// TIA Portal V16 export
// export: Created 2023-03-29T11:03:17.6756957Z, ExportSetting WithDefaults, DisplayName Totally Integrated Automation Portal, DisplayVersion V16 Update 6, DisplayName TIA Portal Version Control Interface, DisplayVersion V16 Update 2, DisplayName TIA Portal Openness, DisplayVersion V16 Update 6, DisplayName STEP 7 Professional, DisplayVersion V16 Update 6, DisplayName STEP 7 Safety, DisplayVersion V16, DisplayName WinCC Advanced, DisplayVersion V16 Update 6
ORGANIZATION_BLOCK "Startup"   // OB100, LAD, Startup
TITLE = "Complete Restart"
{ S7_Optimized_Access := 'TRUE' }
VERSION : 0.1
// Zasuwa status aut. zamknięta= 35980
// Zasuwa status aut. otwarta=34438
// stored: AutoNumber true, IsIECCheckEnabled false, SetENOAutomatically false
   VAR_INPUT
      LostRetentive : Bool;   // True if retentive data are lost
      LostRTC : Bool;   // True if date and time are lost
   END_VAR
BEGIN

REGION Network 1: znacznik powrotu zasilania
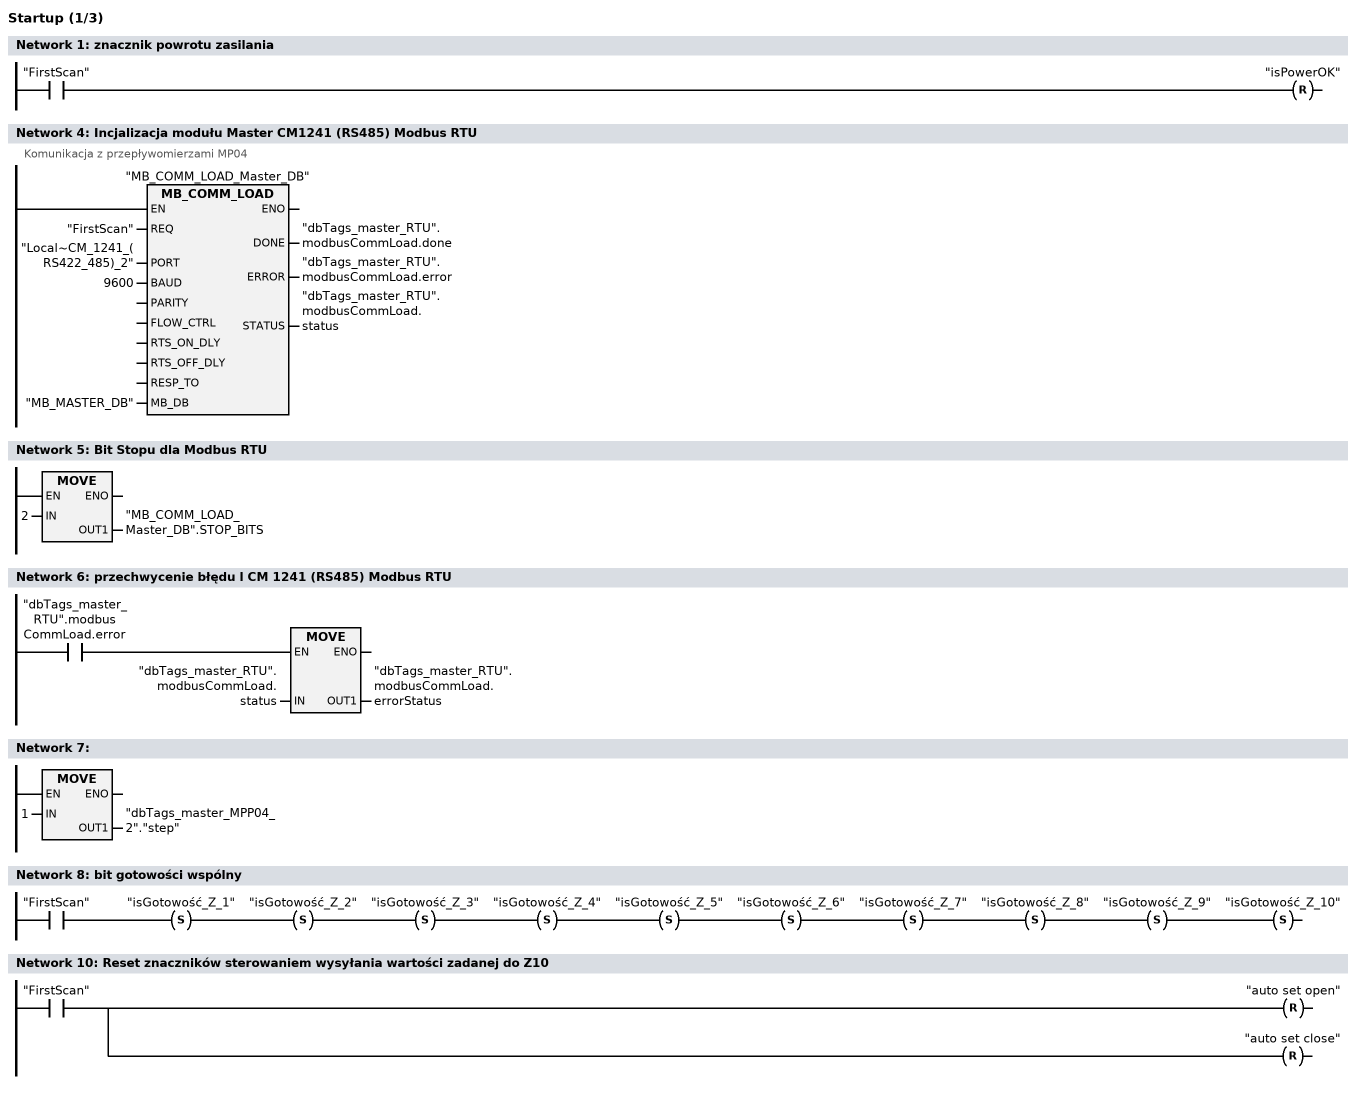
   RUNG wire#powerrail
      Contact( "FirstScan" )
      R_Coil( "isPowerOK" )
   END_RUNG
   // the same network as SCL:
   IF "FirstScan" THEN "isPowerOK" := FALSE; END_IF;
END_REGION

REGION Network 2 (SCL): konfiguracja filtru Kalmana
   IF "FirstScan" THEN //w pierwszym cyklu sterownika
     FOR "I" := 0 TO 3 DO
       "KALMAN_DB".kalman_K["I"] := 0.0;
       "KALMAN_DB".kalman_R["I"] := 0.001;  //niepewność pomiaru
       "KALMAN_DB".kalman_Q["I"] := 0.00001;  //niepewność procesu
       "KALMAN_DB".kalman_P["I"] := 1.0;
     END_FOR;        //parametry R i Q można dobrać osobno dla każdego kanału
   END_IF;           //zostaje wykonana inicjalizacja wszystkich 5 torów analogowych
END_REGION

REGION Network 3 (SCL): Kasowanie alarmów
   "dbtags_Sterowanie".HMI.resetScreen_1 := TRUE;
   "dbtags_Sterowanie".HMI.resetScreen_5 := TRUE;
   "dbtags_Sterowanie".HMI.resetScreen_4 := TRUE;
   "dbtags_Sterowanie".HMI.resetScreen_3 := TRUE;
   "dbtags_Sterowanie".HMI.resetScreen_2 := TRUE;
END_REGION

REGION Network 4: Incjalizacja modułu Master CM1241 (RS485) Modbus RTU
   // Komunikacja z przepływomierzami MP04
   RUNG wire#powerrail
      "MB_COMM_LOAD_Master_DB".MB_COMM_LOAD(REQ := "FirstScan", PORT := "Local~CM_1241_(RS422_485)_2", BAUD := 9600, PARITY :=, FLOW_CTRL :=, RTS_ON_DLY :=, RTS_OFF_DLY :=, RESP_TO :=, MB_DB := "MB_MASTER_DB", DONE => "dbTags_master_RTU".modbusCommLoad.done, ERROR => "dbTags_master_RTU".modbusCommLoad.error, STATUS => "dbTags_master_RTU".modbusCommLoad.status)
   END_RUNG
   // the same network as SCL:
   "MB_COMM_LOAD_Master_DB"(REQ := "FirstScan",   // MB_COMM_LOAD
                           PORT := "Local~CM_1241_(RS422_485)_2",
                           BAUD := 9600,
                           MB_DB := "MB_MASTER_DB",
                           DONE => "dbTags_master_RTU".modbusCommLoad.done,
                           ERROR => "dbTags_master_RTU".modbusCommLoad.error,
                           STATUS => "dbTags_master_RTU".modbusCommLoad.status);
END_REGION

REGION Network 5: Bit Stopu dla Modbus RTU
   RUNG wire#powerrail
      Move(in := 2, out1 => "MB_COMM_LOAD_Master_DB".STOP_BITS)
   END_RUNG
   // the same network as SCL:
   "MB_COMM_LOAD_Master_DB".STOP_BITS := 2;
END_REGION

REGION Network 6: przechwycenie błędu l CM 1241 (RS485) Modbus RTU
   RUNG wire#powerrail
      Contact( "dbTags_master_RTU".modbusCommLoad.error )
      { S7_GenerateENO := "TRUE" } Move(in := "dbTags_master_RTU".modbusCommLoad.status, out1 => "dbTags_master_RTU".modbusCommLoad.errorStatus)
   END_RUNG
   // the same network as SCL:
   IF "dbTags_master_RTU".modbusCommLoad.error THEN
       "dbTags_master_RTU".modbusCommLoad.errorStatus := "dbTags_master_RTU".modbusCommLoad.status;
   END_IF;
END_REGION

REGION Network 7
   RUNG wire#powerrail
      Move(in := 1, out1 => "dbTags_master_MPP04_2"."step")
   END_RUNG
   // the same network as SCL:
   "dbTags_master_MPP04_2"."step" := 1;
END_REGION

REGION Network 8: bit gotowości wspólny
   RUNG wire#powerrail
      Contact( "FirstScan" )
      S_Coil( "isGotowość_Z_1" )
      S_Coil( "isGotowość_Z_2" )
      S_Coil( "isGotowość_Z_3" )
      S_Coil( "isGotowość_Z_4" )
      S_Coil( "isGotowość_Z_5" )
      S_Coil( "isGotowość_Z_6" )
      S_Coil( "isGotowość_Z_7" )
      S_Coil( "isGotowość_Z_8" )
      S_Coil( "isGotowość_Z_9" )
      S_Coil( "isGotowość_Z_10" )
   END_RUNG
   // the same network as SCL:
   IF "FirstScan" THEN
       "isGotowość_Z_1" := TRUE;
       "isGotowość_Z_2" := TRUE;
       "isGotowość_Z_3" := TRUE;
       "isGotowość_Z_4" := TRUE;
       "isGotowość_Z_5" := TRUE;
       "isGotowość_Z_6" := TRUE;
       "isGotowość_Z_7" := TRUE;
       "isGotowość_Z_8" := TRUE;
       "isGotowość_Z_9" := TRUE;
       "isGotowość_Z_10" := TRUE;
   END_IF;
END_REGION

REGION Network 9 (SCL): Wysanie paremetrów sterowania i konfigyracji
     // przekazanie  danych

     "DB10_instance_SCADA".setPołożenieZ10 := "Parametryzacja"."Setting Controll".setPołożenieZ10;
     "DB10_instance_SCADA".ModelSterowania := "Parametryzacja"."Setting Controll".ModelSterowania;
     "DB10_instance_SCADA".TrybSterowania := "Parametryzacja"."Setting Controll".TrybSterowania;
     "DB10_instance_SCADA".setPoziomNapełniania := "Parametryzacja"."Setting Controll".setPoziomNapełniania;
     "DB10_instance_SCADA".setPoziomOpróżnianai := "Parametryzacja"."Setting Controll".setPoziomOpróżnianai;
     // status zasuw
     "DB10_instance_SCADA".instZ1 := "Parametryzacja"."Status drivers".instZ1;
     "DB10_instance_SCADA".instZ2 := "Parametryzacja"."Status drivers".instZ2;
     "DB10_instance_SCADA".instZ3 := "Parametryzacja"."Status drivers".instZ3;
     "DB10_instance_SCADA".instZ4 := "Parametryzacja"."Status drivers".instZ4;
     "DB10_instance_SCADA".instZ5 := "Parametryzacja"."Status drivers".instZ5;
     "DB10_instance_SCADA".instZ6 := "Parametryzacja"."Status drivers".instZ6;
     "DB10_instance_SCADA".instZ7 := "Parametryzacja"."Status drivers".instZ7;
     "DB10_instance_SCADA".instZ8 := "Parametryzacja"."Status drivers".instZ8;
     "DB10_instance_SCADA".instZ9 := "Parametryzacja"."Status drivers".instZ9;
     "DB10_instance_SCADA".instZ10 := "Parametryzacja"."Status drivers".instZ10;

     "DB10_instance_SCADA".actDTL_FillingOn:= "Parametryzacja"."Time Tanks".Start_napełnianie;
     "DB10_instance_SCADA".actDTL_FillingOff:= "Parametryzacja"."Time Tanks".Stop_napełnianie ;
     "DB10_instance_SCADA".actDTL_pumpingOn:= "Parametryzacja"."Time Tanks".Start_przetłaczanie_1 ;
     "DB10_instance_SCADA".actDTL_pumpingOff:= "Parametryzacja"."Time Tanks".Stop_przetłaczanie_1 ;
     "DB10_instance_SCADA".actDTL_RechargingOn:= "Parametryzacja"."Time Tanks".Start_dosilanie_1 ;
     "DB10_instance_SCADA".actDTL_RechargingOff:= "Parametryzacja"."Time Tanks".Stop_dosilanie_1 ;

     "ProcessMemory_Static_1_setChanging" := FALSE;
END_REGION

REGION Network 10: Reset znaczników sterowaniem wysyłania wartości zadanej do Z10
   RUNG wire#powerrail
      Contact( "FirstScan" )
      wire#w1
      R_Coil( "auto set open" )
   END_RUNG
   RUNG wire#w1
      R_Coil( "auto set close" )
   END_RUNG
   // the same network as SCL:
   IF "FirstScan" THEN
       "auto set open" := FALSE;
       "auto set close" := FALSE;
   END_IF;
END_REGION

REGION Network 11: Inicjacja kolejności wywołania Modbus TCP
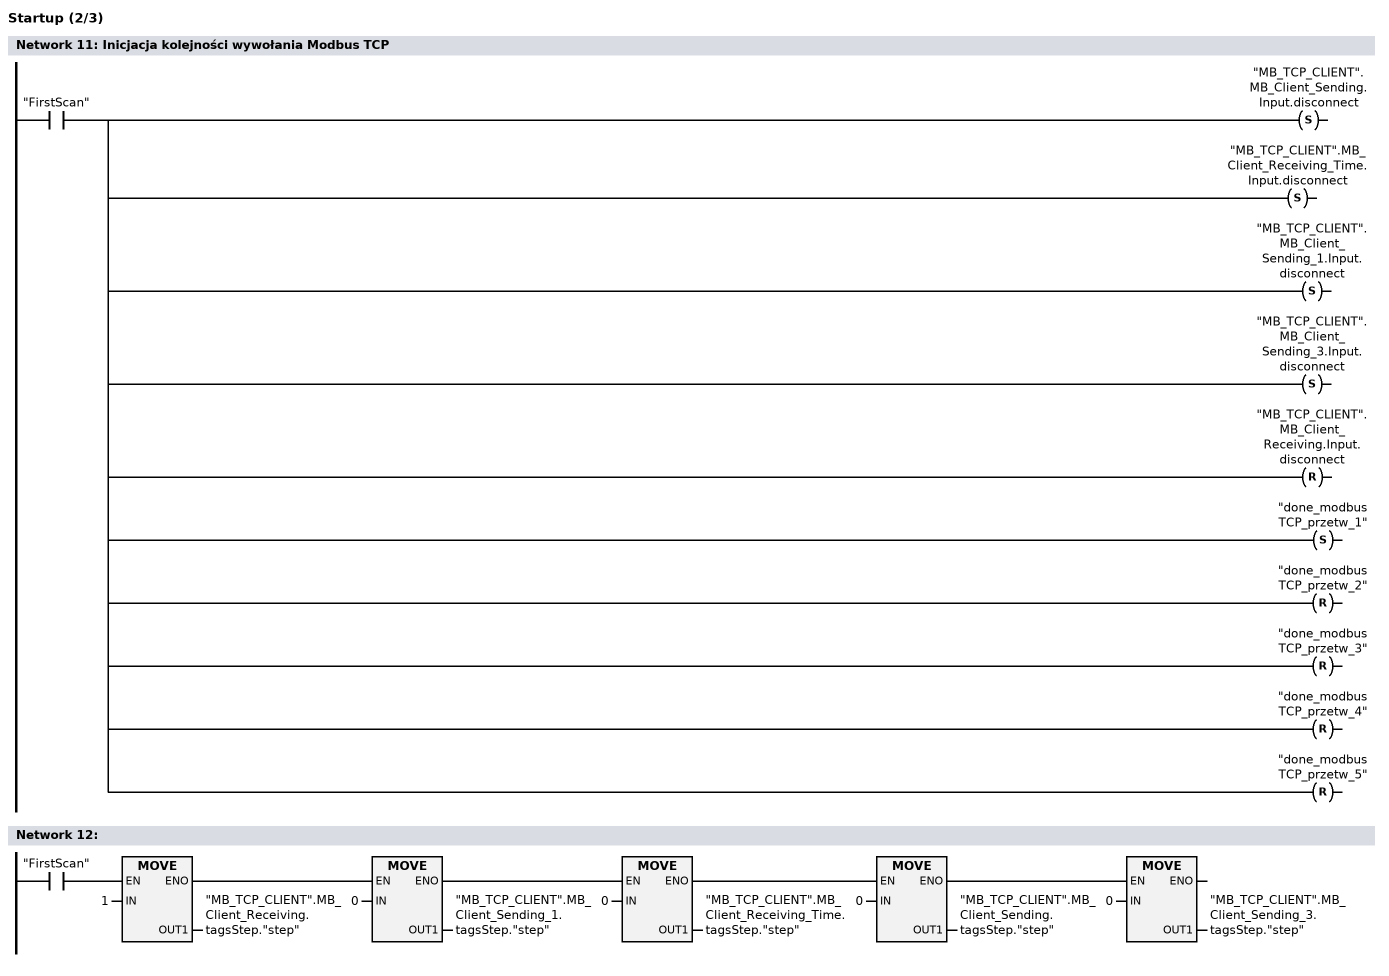
   RUNG wire#powerrail
      Contact( "FirstScan" )
      wire#w1
      S_Coil( "MB_TCP_CLIENT".MB_Client_Sending.Input.disconnect )
   END_RUNG
   RUNG wire#w1
      S_Coil( "MB_TCP_CLIENT".MB_Client_Receiving_Time.Input.disconnect )
   END_RUNG
   RUNG wire#w1
      S_Coil( "MB_TCP_CLIENT".MB_Client_Sending_1.Input.disconnect )
   END_RUNG
   RUNG wire#w1
      S_Coil( "MB_TCP_CLIENT".MB_Client_Sending_3.Input.disconnect )
   END_RUNG
   RUNG wire#w1
      R_Coil( "MB_TCP_CLIENT".MB_Client_Receiving.Input.disconnect )
   END_RUNG
   RUNG wire#w1
      S_Coil( "done_modbusTCP_przetw_1" )
   END_RUNG
   RUNG wire#w1
      R_Coil( "done_modbusTCP_przetw_2" )
   END_RUNG
   RUNG wire#w1
      R_Coil( "done_modbusTCP_przetw_3" )
   END_RUNG
   RUNG wire#w1
      R_Coil( "done_modbusTCP_przetw_4" )
   END_RUNG
   RUNG wire#w1
      R_Coil( "done_modbusTCP_przetw_5" )
   END_RUNG
   // the same network as SCL:
   IF "FirstScan" THEN
       "MB_TCP_CLIENT".MB_Client_Sending.Input.disconnect := TRUE;
       "MB_TCP_CLIENT".MB_Client_Receiving_Time.Input.disconnect := TRUE;
       "MB_TCP_CLIENT".MB_Client_Sending_1.Input.disconnect := TRUE;
       "MB_TCP_CLIENT".MB_Client_Sending_3.Input.disconnect := TRUE;
       "MB_TCP_CLIENT".MB_Client_Receiving.Input.disconnect := FALSE;
       "done_modbusTCP_przetw_1" := TRUE;
       "done_modbusTCP_przetw_2" := FALSE;
       "done_modbusTCP_przetw_3" := FALSE;
       "done_modbusTCP_przetw_4" := FALSE;
       "done_modbusTCP_przetw_5" := FALSE;
   END_IF;
END_REGION

REGION Network 12
   RUNG wire#powerrail
      Contact( "FirstScan" )
      Move(in := 1, out1 => "MB_TCP_CLIENT".MB_Client_Receiving.tagsStep."step")
      Move(in := 0, out1 => "MB_TCP_CLIENT".MB_Client_Sending_1.tagsStep."step")
      Move(in := 0, out1 => "MB_TCP_CLIENT".MB_Client_Receiving_Time.tagsStep."step")
      Move(in := 0, out1 => "MB_TCP_CLIENT".MB_Client_Sending.tagsStep."step")
      Move(in := 0, out1 => "MB_TCP_CLIENT".MB_Client_Sending_3.tagsStep."step")
   END_RUNG
   // the same network as SCL:
   IF "FirstScan" THEN
       "MB_TCP_CLIENT".MB_Client_Receiving.tagsStep."step" := 1;
       "MB_TCP_CLIENT".MB_Client_Sending_1.tagsStep."step" := 0;
       "MB_TCP_CLIENT".MB_Client_Receiving_Time.tagsStep."step" := 0;
       "MB_TCP_CLIENT".MB_Client_Sending.tagsStep."step" := 0;
       "MB_TCP_CLIENT".MB_Client_Sending_3.tagsStep."step" := 0;
   END_IF;
END_REGION

REGION Network 13
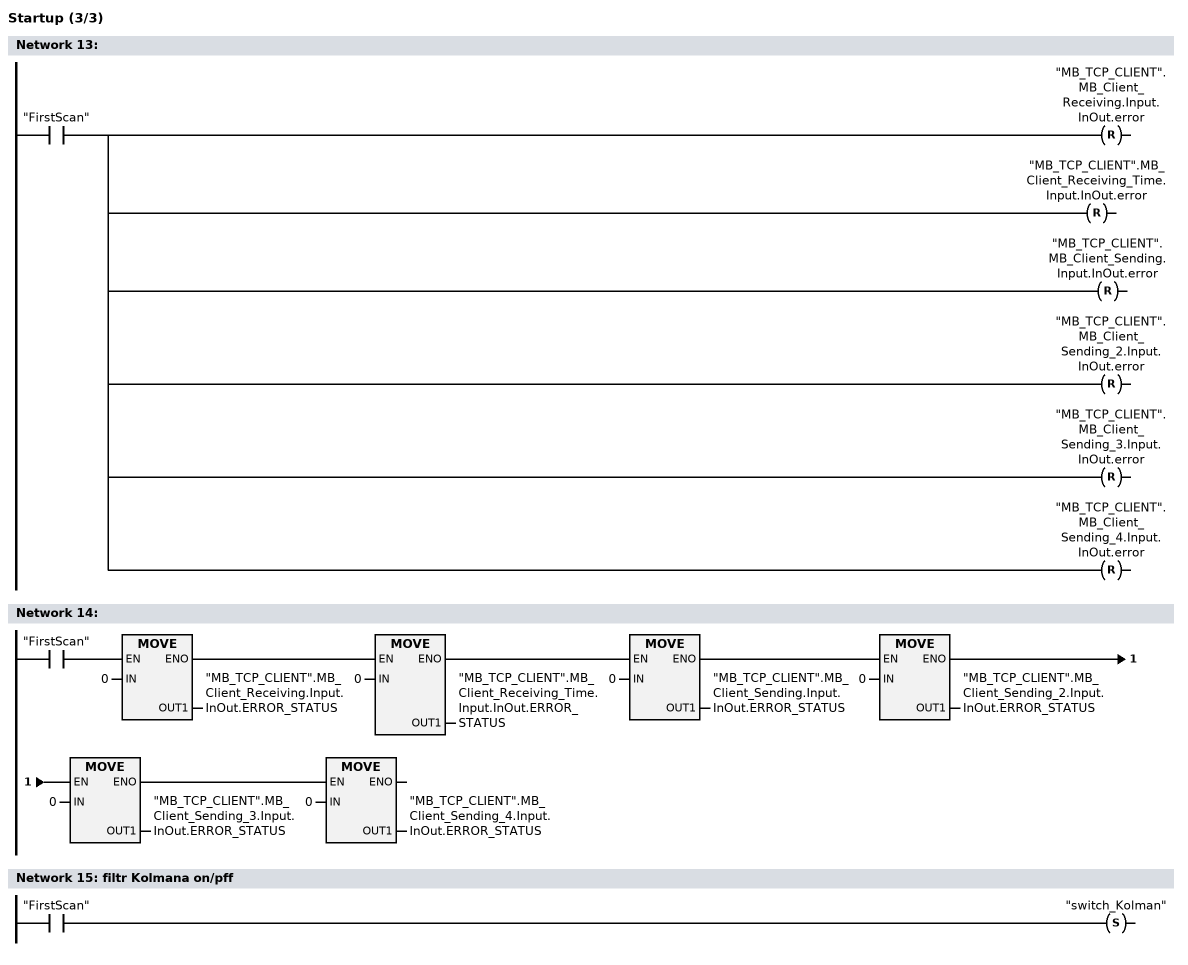
   RUNG wire#powerrail
      Contact( "FirstScan" )
      wire#w1
      R_Coil( "MB_TCP_CLIENT".MB_Client_Receiving.Input.InOut.error )
   END_RUNG
   RUNG wire#w1
      R_Coil( "MB_TCP_CLIENT".MB_Client_Receiving_Time.Input.InOut.error )
   END_RUNG
   RUNG wire#w1
      R_Coil( "MB_TCP_CLIENT".MB_Client_Sending.Input.InOut.error )
   END_RUNG
   RUNG wire#w1
      R_Coil( "MB_TCP_CLIENT".MB_Client_Sending_2.Input.InOut.error )
   END_RUNG
   RUNG wire#w1
      R_Coil( "MB_TCP_CLIENT".MB_Client_Sending_3.Input.InOut.error )
   END_RUNG
   RUNG wire#w1
      R_Coil( "MB_TCP_CLIENT".MB_Client_Sending_4.Input.InOut.error )
   END_RUNG
   // the same network as SCL:
   IF "FirstScan" THEN
       "MB_TCP_CLIENT".MB_Client_Receiving.Input.InOut.error := FALSE;
       "MB_TCP_CLIENT".MB_Client_Receiving_Time.Input.InOut.error := FALSE;
       "MB_TCP_CLIENT".MB_Client_Sending.Input.InOut.error := FALSE;
       "MB_TCP_CLIENT".MB_Client_Sending_2.Input.InOut.error := FALSE;
       "MB_TCP_CLIENT".MB_Client_Sending_3.Input.InOut.error := FALSE;
       "MB_TCP_CLIENT".MB_Client_Sending_4.Input.InOut.error := FALSE;
   END_IF;
END_REGION

REGION Network 14
   RUNG wire#powerrail
      Contact( "FirstScan" )
      Move(in := 0, out1 => "MB_TCP_CLIENT".MB_Client_Receiving.Input.InOut.ERROR_STATUS)
      Move(in := 0, out1 => "MB_TCP_CLIENT".MB_Client_Receiving_Time.Input.InOut.ERROR_STATUS)
      Move(in := 0, out1 => "MB_TCP_CLIENT".MB_Client_Sending.Input.InOut.ERROR_STATUS)
      Move(in := 0, out1 => "MB_TCP_CLIENT".MB_Client_Sending_2.Input.InOut.ERROR_STATUS)
      Move(in := 0, out1 => "MB_TCP_CLIENT".MB_Client_Sending_3.Input.InOut.ERROR_STATUS)
      Move(in := 0, out1 => "MB_TCP_CLIENT".MB_Client_Sending_4.Input.InOut.ERROR_STATUS)
   END_RUNG
   // the same network as SCL:
   IF "FirstScan" THEN
       "MB_TCP_CLIENT".MB_Client_Receiving.Input.InOut.ERROR_STATUS := 0;
       "MB_TCP_CLIENT".MB_Client_Receiving_Time.Input.InOut.ERROR_STATUS := 0;
       "MB_TCP_CLIENT".MB_Client_Sending.Input.InOut.ERROR_STATUS := 0;
       "MB_TCP_CLIENT".MB_Client_Sending_2.Input.InOut.ERROR_STATUS := 0;
       "MB_TCP_CLIENT".MB_Client_Sending_3.Input.InOut.ERROR_STATUS := 0;
       "MB_TCP_CLIENT".MB_Client_Sending_4.Input.InOut.ERROR_STATUS := 0;
   END_IF;
END_REGION

REGION Network 15: filtr Kolmana on/pff
   RUNG wire#powerrail
      Contact( "FirstScan" )
      S_Coil( "switch_Kolman" )
   END_RUNG
   // the same network as SCL:
   IF "FirstScan" THEN "switch_Kolman" := TRUE; END_IF;
END_REGION
END_ORGANIZATION_BLOCK
